Universal Robots PolyScope program: step5c_joint_rnn_cycloid_v1.urp

Program step5c_joint_rnn_cycloid_v1 (installation=default directory=/programs/andyl/kunwei/step5 createdIn=5.11.9.1010452 lastSavedIn=5.11.9.1010452 robotSerialNumber=20225200364)
Calibrated DH parameters: a=[0.00002, -0.569483, -0.54992, -0.00001, -0.000036, 0]; d=[0.180894, -146.691669, 192.918669, -46.053088, 0.119778, 0.115602]; alpha=[1.571425, -0.001534, 0.003359, 1.568739, -1.571477, 0]; deltaTheta=[0, 0.376258, -0.101074, -0.275185, -0.000002, 0]
Robot Program (runOnlyOnce=true)
  Script file /programs/andyl/kunwei/step5/step5c_joint_rnn_cycloid_v1.script
    | # Step5c joint-RNN contact quarantine.
    | # VERSION: 2026-06-13T0041HKT_STEP5C_JOINT_RNN_CYCLOID_V1
    | # GENERATED_AT_LOCAL: 2026-06-13T00:41:36+08:00
    | # FLOW_TABLE: STEP5_FLOW.md
    | # STEP5_STAGE_ID: step5c_joint_rnn_cycloid_v1
    | # STEP5_TABLE_SOURCE: config/step5_stage_table.json
    | # QUARANTINE_REASON: previous package was bounded DLS/IK, not strict TASE RNN; contact is blocked.
    | # TP_ROLE: stop_only_quarantine; no motion command, no contact search, no bridge command consumption.
    | # SAFETY: no speedj, no speedl, no force_mode, no zero_ftsensor(), no TCP/payload write.
    | 
    | def codex_step5c_joint_rnn_cycloid_v1():
    |   textmsg("codex step5c contact quarantine 2026-06-13T0041HKT_STEP5C_JOINT_RNN_CYCLOID_V1: strict RNN not implemented; refusing motion")
    |   write_output_float_register(30, 91.0)
    |   write_output_float_register(31, 0.0)
    |   write_output_float_register(35, 29.0)
    | end
    | 
    | codex_step5c_joint_rnn_cycloid_v1()
